FUNCTION_BLOCK FB_CommandChangeUnSuspend EXTENDS FB_CommandChange IMPLEMENTS ITF_CommandChange
VAR

END_VAR

(*			
	RafalOS
	Rafał Osajda		03.11.2025		TC 4024.66
	Test czy można zmienić stan lub tryb i zwraca czy można i uruchamia zmianę
*)
METHOD PUBLIC Execute : BOOL
VAR_INPUT
	iNumberOfCommand	: INT;
END_VAR
IF (THIS^.itfSaMController.GetState () = E_BaseMachineState.Suspended) THEN		// sprawdzenie czy jesteśmy w dobrym stanie dla tego rozkazu
	IF (THIS^.itfSaMController.IsStateInModeEnabled (eNewState := E_BaseMachineState.Unsuspending)) THEN	//test czy stan do którego chcemy przejśc jest właczony dla tego trybu
		THIS^.itfSaMController.ChangeStateTo (eNewState := E_BaseMachineState.Unsuspending);
	ELSE
		THIS^.EventSetActive (iNumber := 5);	//stan docelowy jest wylaczony w tym trybie
	END_IF
ELSE
	THIS^.EventSetActive (iNumber := 4);	//ten rozkaz nie obsluguje tego stanu
END_IF
END_METHOD

METHOD FB_init : BOOL
VAR_INPUT
	bInitRetains : BOOL; // if TRUE, the retain variables are initialized (warm start / cold start)
	bInCopyCode : BOOL;  // if TRUE, the instance afterwards gets moved into the copy code (online change)
END_VAR
THIS^.SetText (eLocation := E_BaseLocation.pl, wsDescription := "Command change state - UnSuspend");
THIS^.SetText (eLocation := E_BaseLocation.en, wsDescription := "Command change state - UnSuspend");
THIS^.SetText (eLocation := E_BaseLocation.de, wsDescription := "Command change state - UnSuspend");
THIS^.SetName (stName := THIS^.GetTexts ());
END_METHOD

END_FUNCTION_BLOCK

(* stored: Version 1.1.0.1
   POU FB_CommandChangeUnSuspend: Id {03c9589a-fc15-0c4a-14e8-fb8dbfc85e4c}, SpecialFunc None
   Method Execute: Id {4e3cd498-9382-0c9e-342c-b96d044b02bb}
   Method FB_init: Id {c514234a-21b6-0e57-069f-5aa61bb04c72} *)
